// Copyright (c) 2024 Loupe (https://loupe.team), provided under the MIT License.
{attribute 'qualified_only'}
{attribute 'strict'}
TYPE ABBLINKIN_DATA_TYPE_Typ :
(
	_NONE,
	_STRING,
	_BOOL,
	_DINT,
	_LREAL
);
END_TYPE

(* stored: Version 1.1.0.1, ProductVersion 3.1.4024.12
   DUT ABBLINKIN_DATA_TYPE_Typ: Id {ab428c6a-3178-4506-83fd-90df6da75be6} *)
